TYPE UDT_ProgramStatus_RD :
STRUCT
 
error : BOOL; // 有错误
errorID : Word; // 错误代码
errorText : String[100]; // 错误文本信息
warning : Bool; // 有警告
warnID : Word; // 警告代码
warnText : String[100]; // 警告文本信息
  
END_STRUCT
END_TYPE

(* stored: Version 1.1.0.1, ProductVersion 3.1.4024.12
   DUT UDT_ProgramStatus_RD: Id {ad655455-24b0-4298-ae8b-638f6a386d11} *)
